// TIA Portal V19 export
DATA_BLOCK "Loop1_PERS"   // DB194
{ DB_Accessible_From_OPC_UA := 'FALSE' }
// stored: DBAccessibleFromOPCUA false, MemoryReserve 100
   VAR RETAIN
      PersistentValues : Struct
         Par { S7_SetPoint := 'True'} : "SmartLoopControl_Par";
      END_STRUCT;
   END_VAR
   VAR
      AuxPE_LsMax_TP_Entry : Bool := FALSE;
      AuxPE_LsMax_TP_Exit : Bool := FALSE;
   END_VAR
BEGIN
   PersistentValues.Par.WorkMode := 1;
   PersistentValues.Par.SyncEntryMode := 0;
   PersistentValues.Par.SyncExitMode := 0;
   PersistentValues.Par.PosStopMinHigh := 19200.0;
   PersistentValues.Par.PosStopMiddle := 19550.0;
   PersistentValues.Par.PosStopMaxLow := 19836.0;
   PersistentValues.Par.PosSynch := 19836.0;
   PersistentValues.Par.PosDeltaRestartAfterMaxLow := 5.0;
   PersistentValues.Par.PosDeltaRestartAfteMinHigh := 200.0;
   PersistentValues.Par.PosIntervalSynchroCyclic := 500000.0;
   PersistentValues.Par.HysteresysSynchroExt := 5000.0;
   PersistentValues.Par.Entry_Lim1_VMin := 50.0;
   PersistentValues.Par.Entry_Lim2_VMed := 100.0;
   PersistentValues.Par.Entry_Lim3_VMax := 150.0;
   PersistentValues.Par.Entry_Override1_VMin := 10.0;
   PersistentValues.Par.Entry_Override2_VMed := 95.0;
   PersistentValues.Par.Entry_Override3_VMax := 105.0;
   PersistentValues.Par.Exit_Lim1_VMin := 100.0;
   PersistentValues.Par.Exit_Lim2_VMed := 200.0;
   PersistentValues.Par.Exit_Lim3_VMax := 400.0;
   PersistentValues.Par.Exit_Override1_VMin := 10.0;
   PersistentValues.Par.Exit_Override2_VMed := 100.0;
   PersistentValues.Par.Exit_Override3_VMax := 100.0;
   PersistentValues.Par.DlySetMaxLow := T#500MS;
   PersistentValues.Par.DlyRstMaxLow := T#500MS;
   PersistentValues.Par.Exit_MaxFeed_CaseSystemOff := 300.0;
   PersistentValues.Par.Exit_MaxFeed_CaseNextEndOfMaterial := 300.0;
   PersistentValues.Par.Exit_MaxFeed_CaseLoopMaterialNotValid := 200.0;
END_DATA_BLOCK
